PROGRAM S01_Loading
VAR
	//工站
	station					: REFERENCE TO FB_Station:=fbstation[1];
	//气缸
		fbVTCPressCyl_1	:REFERENCE TO FB_Cylinder:=fbCylinder[1];	//	链板线-下压气缸1
		fbVTCPressCyl_2	:REFERENCE TO FB_Cylinder:=fbCylinder[2];	//	链板线-下压气缸2
		fbVTCPressCyl_3	:REFERENCE TO FB_Cylinder:=fbCylinder[3];	//	链板线-下压气缸3
		fbVTCPressCyl_4	:REFERENCE TO FB_Cylinder:=fbCylinder[4];	//	链板线-下压气缸4
		fbVTCCyl_1	:REFERENCE TO FB_Cylinder:=fbCylinder[5];	//	移栽机构-Z轴气缸1
		fbVTCCyl_2	:REFERENCE TO FB_Cylinder:=fbCylinder[6];	//	移栽机构-Z轴气缸2
//链板线
		fbFlowLine:FB_FlowLine;	
		
	//伺服
		fbXAxisMove	 :REFERENCE TO FB_Axis:=fbAxis[1];	//	移栽上料X轴伺服
		fbYAxisMove	 :REFERENCE TO FB_Axis:=fbAxis[2];	//	移栽上料Y轴伺服
	//电动夹爪
		fbClamp_1:	 REFERENCE TO FB_ERG_20_Modbus:=fbERG_20_Modbus[1];
		fbClamp_2:	 REFERENCE TO FB_ERG_20_Modbus:=fbERG_20_Modbus[2];
	//相机
		 Camera   : 	 REFERENCE TO FB_Camera:=fbCamera[1]; 
	//延时
	arTonDelay :ARRAY[1..20] OF TON;
	//返回值
	UdiReturnValue :ARRAY[1..20] OF UDINT;
	//本地过程数据
	arProcessDataStation : ARRAY [1..2] OF DUT_MainlineFixture;
	//过程标志位
	xFlowLineReady:BOOL;//连班线准备流程完成信号
	xTakeBoxPremit:BOOL;//允许链板线执行下一循环
	//过程记录
	tsModuleProcess:ARRAY[1..gc_ModuleProNo] OF DUT_Process;
	xClearModuleProcessDone:BOOL;
	bClearProcessStep	:BYTE;
	
	
	i: INT;
	xFlowLineStart: BOOL;//链板线启动信号
	bFlowLineStep: BYTE;
	xFlowLineReadyCmd: BOOL;//连班线准备指令
	arFlowLineReachedSensor: ARRAY[1..4] OF BOOL;//链板线到位传感器
	_FirstFlag: ARRAY[1..10] OF BOOL;
	MachineInitR_TRIG:R_TRIG;

	// 程序循环
	bCounter: BYTE;
	// 上料工位到位传感器
	xLoadingReachedSensor: ARRAY[1..2] of bool;
	// 报警标志位
	_AlarmDisable: BOOL;
	// X轴放料循环
	bXCounter: BYTE;
	//夹爪有产品信号
	arClampHavePart :ARRAY[1..2] OF BOOL;
	iClearProcessStep: INT;
	// //首次循环
	_FirstCycle: ARRAY[1..10] of bool;
	//下压气缸原点传感器
	arVTCPressCylHPSensor:ARRAY[1..4] OF BOOL;
	//Y轴去放料位还是放料补偿位
	ariPosNum:ARRAY[1..2] OF INT;
	//下压气缸动点传感器
	arVTCPressCylWPSensor:ARRAY[1..4] OF BOOL;
	test: ARRAY[1..4]OF BOOL;
END_VAR

A_Input();
Alarm();
Delay();
FlowAuto();
FlowInit();
FlowLine();
General();
ILC();
TipAuto();
TipManual();
Z_Output();

ACTION A_Input:
//气缸
fbVTCPressCyl_1.xWP_Sensor	:=
arVTCPressCylWPSensor[1]		:=	IxS01VTCPressCyl_1WP 	;
fbVTCPressCyl_1.xHP_Sensor	:=
arVTCPressCylHPSensor[1]		:=	IxS01VTCPressCyl_1HP	;
fbVTCPressCyl_2.xWP_Sensor	:=	
arVTCPressCylWPSensor[2]		:=	IxS01VTCPressCyl_2WP	;
fbVTCPressCyl_2.xHP_Sensor	:=
arVTCPressCylHPSensor[2]		:=	IxS01VTCPressCyl_2HP	;
fbVTCPressCyl_3.xWP_Sensor	:=	
arVTCPressCylWPSensor[3]		:=IxS01VTCPressCyl_3WP	;
fbVTCPressCyl_3.xHP_Sensor	:=
arVTCPressCylHPSensor[3]		:=	IxS01VTCPressCyl_3HP	;
fbVTCPressCyl_4.xWP_Sensor	:=	
arVTCPressCylWPSensor[4]		:=IxS01VTCPressCyl_4WP	;
fbVTCPressCyl_4.xHP_Sensor	:=
arVTCPressCylHPSensor[4]		:=IxS01VTCPressCyl_4HP	;
fbVTCCyl_1.xWP_Sensor	:=	IxS01VTCCyl_1WP	;
fbVTCCyl_1.xHP_Sensor	:=	IxS01VTCCyl_1HP	;
fbVTCCyl_2.xWP_Sensor	:=	IxS01VTCCyl_2WP	;
fbVTCCyl_2.xHP_Sensor	:=	IxS01VTCCyl_2HP	;

//链板线传感器
arFlowLineReachedSensor[1]:=IxS01PositionSensor2;
arFlowLineReachedSensor[2]:=IxS01PositionSensor1;
arFlowLineReachedSensor[3]:=IxS01PositionSensor4;
arFlowLineReachedSensor[4]:=IxS01PositionSensor3;
//上料工位传感器
xLoadingReachedSensor[1]:=IxS01Sensor2Reached;
xLoadingReachedSensor[2]:=IxS01Sensor1Reached;
END_ACTION

ACTION Alarm:
//
station.adwAlarm[1].00:=station.xInitTimeout;	  //S01 初始化超时
(*station.adwAlarm[1].01:= //S01链板线上料位置1相机检测到深孔板放反，请检查
station.adwAlarm[1].02:=//S01链板线上料位置2相机检测到深放反，请检查
station.adwAlarm[1].03:=//S01链板线上料位置3相机检测到深孔板放反，请检查
station.adwAlarm[1].04:=//S01链板线上料位置4相机检测到深孔板放反，请检查
*)
station.adwAlarm[1].05	:=	fbClamp_1.eErrorID>24	;//	S01电动夹爪1报错，请检查
station.adwAlarm[1].06	:=	fbClamp_2.eErrorID>24	;//	S01电动夹爪2报错，请检查
//station.adwAlarm[1].07	:=	fbVTCPressCyl_1.xHP_Off 	;//	S01链板线-下压气缸1原点未到位
//station.adwAlarm[1].08	:=	fbVTCPressCyl_1.xWP_Off 	;//	S01链板线-下压气缸1动点未到位
//station.adwAlarm[1].09	:=	fbVTCPressCyl_2.xHP_Off	;//	S01链板线-下压气缸2原点未到位
//station.adwAlarm[1].10	:=	fbVTCPressCyl_2.xWP_Off	;//	S01链板线-下压气缸2动点未到位
//station.adwAlarm[1].11	:=	fbVTCPressCyl_3.xHP_Off	;//	S01链板线-下压气缸3原点未到位
//station.adwAlarm[1].12	:=	fbVTCPressCyl_3.xWP_Off	;//	S01链板线-下压气缸3动点未到位
//station.adwAlarm[1].13	:=	fbVTCPressCyl_4.xHP_Off	;//	S01链板线-下压气缸4原点未到位
//station.adwAlarm[1].14	:=	fbVTCPressCyl_4.xWP_Off	;//	S01链板线-下压气缸4动点未到位
station.adwAlarm[1].15	:=	fbVTCCyl_1.xHP_Off 	;//	S01移栽机构-Z轴气缸1原点未到位
station.adwAlarm[1].16	:=	fbVTCCyl_1.xWP_Off	;//	S01移栽机构-Z轴气缸1动点未到位
station.adwAlarm[1].17	:=	fbVTCCyl_2.xHP_Off 	;//	S01移栽机构-Z轴气缸2原点未到位
station.adwAlarm[1].18	:=	fbVTCCyl_2.xWP_Off	;//	S01移栽机构-Z轴气缸2动点未到位
station.adwAlarm[1].19	:=	fbXAxisMove.xError	;//	S01移栽上料X轴伺服报错
station.adwAlarm[1].20	:=	fbXAxisMove.xNotPowerOn	;//	S01移栽上料X轴伺服未使能
station.adwAlarm[1].21	:=	fbXAxisMove.xMoveTimeout	;//	S01移栽上料X轴伺服移动超时
station.adwAlarm[1].22	:=	fbYAxisMove.xError	;//	S01移栽上料Y轴伺服报错
station.adwAlarm[1].23	:=	fbYAxisMove.xNotPowerOn	;//	S01移栽上料Y轴伺服未使能
station.adwAlarm[1].24	:=	fbYAxisMove.xMoveTimeout	;//	S01移栽上料Y轴伺服移动超时
//station.adwAlarm[1].25	:=	fbFlowLine.xQError	;			//	S01移栽上料链板线报错

(*station.adwAlarm[1].26:= //S01链板线上料位置1相机检测到深孔板放反，请检查
station.adwAlarm[1].27:=//S01链板线上料位置2相机检测到深放反，请检查
station.adwAlarm[1].28:=//S01链板线上料位置3相机检测到深孔板放反，请检查
station.adwAlarm[1].29:=//S01链板线上料位置4相机检测到深孔板放反，请检查
*)
END_ACTION

ACTION Delay:
arTonDelay[01](IN:= , PT:=T#0.1S , Q=> , ET=> );
(*arTonDelay[02](IN:=  , PT:=T#1S , Q=> , ET=> );*)//链板线程序使用
arTonDelay[03](IN:=   , PT:=T#1S , Q=> , ET=> );
arTonDelay[04](IN:= , PT:=T#0.1S , Q=> , ET=> );
arTonDelay[05](IN:= , PT:=T#0.1S , Q=> , ET=> );
arTonDelay[06](IN:= , PT:=T#0.1S , Q=> , ET=> );
arTonDelay[07](IN:= , PT:=T#0.1S , Q=> , ET=> );
arTonDelay[08](IN:= NOT fbXAxisMove.xbusy , PT:=T#0.1S , Q=> , ET=> );//TipAuto使用
arTonDelay[09](IN:= NOT fbYAxisMove.xbusy, PT:=T#0.1S , Q=> , ET=> );//TipAuto使用
END_ACTION

ACTION FlowAuto:

//-----------------------------------------初始化是否完成判断----------------------------------------------
IF NOT station.xInitDone THEN
 	station.iStepAuto:=0;
 	station.xDone:=FALSE;
ELSIF station.xRunning  THEN
//-----------------------------------------动作步骤--------------------------------------------------------
CASE station.iStepAuto OF	  
	0: //----Home Step，等待启动----
		IF station.xDisabled 
			AND station.xCanRun 
			AND NOT fbMachine[1].xStopped 
			AND NOT station.xSingleRunning 
		THEN
			station.xDone:=TRUE;
		END_IF
		IF  station.xSingleRunning 
			OR station.xCanRun 
			//AND NOT station.xDone 
			AND NOT station.xDisabled 
			AND NOT fbMachine[1].xStopped
		THEN
			station.xCycleEnable:=TRUE;
			//station.xDone:= FALSE;  
			station.iStepAuto:= 10;
		END_IF
	10://复位
			Camera.xlInit:=TRUE;
			FOR  i:=1 TO  4 BY  1 DO
		 		sCamera_To_Plc.iS01Result[i]:=0;
			END_FOR
			MEMSET(ADR(arProcessDataStation[1]),0,SIZEOF(arProcessDataStation[1]));
			MEMSET(ADR(arProcessDataStation[2]),0,SIZEOF(arProcessDataStation[2]));
		
				 FOR i:=1 TO gc_ModuleProNo BY 1 DO
						 MEMSET(ADR(tsModuleProcess[i]),0,SIZEOF(tsModuleProcess[i]));
				 END_FOR
			station.iStepAuto:= 20;
  	20://此处开始处理上料流程
		station.iStepAuto:= 40;
//	30://Restore_after_Estop_Process1-拍照流程
//			IF  axBypassSignal[1] OR fbMachine[1].xTryRun THEN
//					station.iStepAuto :=110 ;
//			ELSIF tsModuleProcess[1].xProcessNotStarted AND NOT  tsModuleProcess[1].xProcessStarted THEN
//					station.iStepAuto :=40 ; (*process not started*)
//			ELSIF  tsModuleProcess[1].xProcessStarted AND NOT  tsModuleProcess[1].xProcessCompleted THEN
//				 station.iStepAuto :=40 ;(*process started*)
//			ELSIF  tsModuleProcess[1].xProcessCompleted AND NOT tsModuleProcess[1].xQDataCompleted  THEN
//					station.iStepAuto := 100 ;(*process completed*)
//			ELSIF tsModuleProcess[1].xQDataCompleted THEN
//					station.iStepAuto :=110 ;(*Qdata completed *)
//			ELSE    
//					station.iStepAuto :=40; 
//			END_IF
	40://启动链板线
		tsModuleProcess[1].xProcessNotStarted:=TRUE;
		fbFlowLine.xIRunningPremit:=TRUE;
			station.iStepAuto:=45;	
	45://链板线已启动
		IF   fbFlowLine.xQBusy THEN
		 		fbFlowLine.xIRunningPremit:=FALSE;
				station.iStepAuto:=50;	
		END_IF
	50://等待链板线执行结束
		IF 		NOT fbFlowLine.xQBusy THEN
		 		station.iStepAuto:=60;	
		END_IF
	60://Y轴去拍照位置
		fbYAxisMove.xMoveAuto[2]:=TRUE;
		IF  fbYAxisMove.xMoveInPos[2] THEN
		  	 station.iStepAuto:=70;	
		END_IF
	70://相机触发
		tsModuleProcess[1].xProcessStarted:=TRUE;
			Camera.xlTrigger:=TRUE;
			IF    Camera.xQBusy THEN
				Camera.xlTrigger:=FALSE;
				station.iStepAuto:=80;	
			END_IF
	80://等待相机完成
		IF  NOT Camera.xQBusy THEN
			station.iStepAuto:=100;		
		END_IF
		tsModuleProcess[1].xProcessCompleted:=TRUE;
	100://查看相机结果，判断是否料反
		(*位置1*)		
		_AlarmDisable:=FALSE;
		FOR  i:=1 TO 4 BY 1 DO
			IF 	sCamera_TO_Plc.iS01Result[i] >=3 THEN
					station.iStepAuto:=101;
					EXIT;
			ELSIF	i =4 THEN
					station.iStepAuto:=110;
			END_IF
		END_FOR
	101://报警,人工处理后重新拍照
		IF  NOT  _AlarmDisable THEN
					IF   sCamera_TO_Plc.iS01Result[1] =3 (*料反*) THEN
						station.adwAlarm[1].01:=TRUE ;//S01链板线上料位置1相机检测到深孔板放反，请检查
					ELSIF  sCamera_TO_Plc.iS01Result[1] =4 (*无料*) THEN
					 	station.adwAlarm[1].26:=TRUE ;//S01链板线上料位置1相机未检测到深孔板，请检查
					END_IF
					IF   sCamera_TO_Plc.iS01Result[2] =3 (*料反*) THEN
						station.adwAlarm[1].02:=TRUE ;//S01链板线上料位置2相机检测到深孔板放反，请检查
					ELSIF  sCamera_TO_Plc.iS01Result[2] =4 (*无料*) THEN
					 	station.adwAlarm[1].27:=TRUE ;//S01链板线上料位置2相机未检到板，请检查
					END_IF	
					IF   sCamera_TO_Plc.iS01Result[3] =3 (*料反*) THEN
 						station.adwAlarm[1].03:= TRUE;//S01链板线上料位置3相机检测到深孔板放反，请检查
					ELSIF  sCamera_TO_Plc.iS01Result[3] =4 (*无料*) THEN
					 	station.adwAlarm[1].28:=TRUE ;//S01链板线上料位置3相机未检到板，请检查
					END_IF
					IF    sCamera_TO_Plc.iS01Result[4] =3 (*料反*) THEN
 						station.adwAlarm[1].04:= TRUE;//S01链板线上料位置4相机检测到深孔板放反，请检查
					ELSIF  sCamera_TO_Plc.iS01Result[4] =4 (*无料*) THEN
					 	station.adwAlarm[1].29:=TRUE ;//S01链板线上料位置4相机未检到板，请检查
					END_IF
					_AlarmDisable:=TRUE;
		END_IF
			station.iStepAuto:=60;
	110://数据传送完成
			tsModuleProcess[1].xQDataCompleted:=TRUE;
			station.iStepAuto:=150;

///预留复检步骤120-150
	150://开始循环。循环次数=2
		IF NOT  fbMachine[1].xTryRun THEN
				IF  arFlowLineReachedSensor[1] AND arFlowLineReachedSensor[3]   THEN
								bCounter:=1;
								station.iStepAuto :=170; 
				ELSIF arFlowLineReachedSensor[2] AND arFlowLineReachedSensor[4] THEN
								bCounter:=2;
								station.iStepAuto :=170; 
				ELSE
								station.iStepAuto :=999; 
				END_IF
				
		ELSE
				 IF   NOT _FirstFlag[2] THEN
						bCounter:=1;
						_FirstFlag[2]:=TRUE;
				END_IF
		 		station.iStepAuto :=170; 
		END_IF
//	160://Restore_after_Estop_Process2/3 取孔板流程1/2
//			IF  station.xSingleRunning OR fbMachine[1].xTryRun THEN
//					station.iStepAuto :=170; 
//			ELSIF tsModuleProcess[bCounter+1].xProcessNotStarted AND NOT  tsModuleProcess[bCounter+1].xProcessStarted THEN
//					station.iStepAuto :=190 ; (*process not started*)
//			ELSIF  tsModuleProcess[bCounter+1].xProcessStarted AND NOT  tsModuleProcess[bCounter+1].xProcessCompleted THEN
//				 station.iStepAuto :=185 ;(*process started*)
//			ELSIF  tsModuleProcess[bCounter+1].xProcessCompleted AND NOT tsModuleProcess[bCounter+1].xQDataCompleted  THEN
//					station.iStepAuto := 230 ;(*process completed*)
//			ELSE
//					station.iStepAuto :=170; 
//			END_IF
	170://
			tsModuleProcess[bCounter+1].xProcessNotStarted :=TRUE;
			 station.iStepAuto:=190;
//		(***异常处理开始*)
//	185://电动夹爪打开
//			fbClamp_1.aReleaseControl[1]:=TRUE;
//			fbClamp_2.aReleaseControl[1]:=TRUE;
//			IF fbClamp_1.xDone  AND fbClamp_2.xDone   THEN
//					fbClamp_1.xExecute :=FALSE ;
//					fbClamp_2.xExecute:=FALSE;
//					 station.iStepAuto:=166;
//			END_IF	
//	186://Z轴上升
//			fbVTCCyl_1.xAuto:=FALSE;
//			fbVTCCyl_2.xAuto:=FALSE;
//		IF  fbVTCCyl_1.xHP_Delay AND 
//			fbVTCCyl_2.xHP_Delay THEN
//			 station.iStepAuto:=190;		
//		END_IF
//	(***异常处理结束*)			  
	190://XY轴去夹取位置1/2
			fbXAxisMove.xMoveAuto[bCounter +1]:=TRUE;
			fbYAxisMove.xMoveAuto[3]:=TRUE;
			fbClamp_1.aRotateReleaseControl[1]:=TRUE ;
			fbClamp_2.aRotateReleaseControl[1]:=TRUE ;		
			IF fbXAxisMove.xMoveInPos[bCounter+1] AND 
			   fbYAxisMove.xMoveInPos[3] AND 
				 fbClamp_1.xDone AND  
			  fbClamp_2.xDone THEN
					fbClamp_1.xExecute :=FALSE ;
				 fbClamp_2.xExecute :=FALSE ;
				 station.iStepAuto:=200;	
			END_IF
			
	200://Z轴气缸下降
		fbVTCCyl_1.xAuto:=TRUE;
		fbVTCCyl_2.xAuto:=TRUE;
		IF  fbVTCCyl_1.xWP_Delay AND 
			fbVTCCyl_2.xWP_Delay THEN
			 station.iStepAuto:=210;		
		END_IF
	210://电动夹爪夹取
				tsModuleProcess[bCounter+1].xProcessStarted :=TRUE;
		IF  fbmachine[1].xTryRun THEN 
				station.iStepAuto:=220;	
		ELSE
			fbClamp_1.aClampControl[1]:=TRUE;
			fbClamp_2.aClampControl[1]:=TRUE;
			IF (fbClamp_1.xDone OR (fbClamp_1.xGripClampEmpty  AND fbMachine[1].xTryRun)) AND
			 (fbClamp_2.xDone OR (fbClamp_2.xGripClampEmpty  AND fbMachine[1].xTryRun ))   THEN
					fbClamp_1.xExecute :=FALSE ;
					fbClamp_2.xExecute:=FALSE;
					 station.iStepAuto:=220;	
			END_IF
		END_IF	 
	220://Z轴上升
			arClampHavePart[1]:=TRUE;//夹爪1有产品标志位
			arClampHavePart[2]:=TRUE;//夹爪2有产品标志位
			tsModuleProcess[bCounter+1].xProcessCompleted :=TRUE;
				fbVTCCyl_1.xAuto:=FALSE;
				fbVTCCyl_2.xAuto:=FALSE;
			IF  fbVTCCyl_1.xHP_Delay AND 
				fbVTCCyl_2.xHP_Delay THEN
				 station.iStepAuto:=225;		
			END_IF
	225://判断流程
			IF bCounter =2 THEN
					xTakeBoxPremit:=TRUE;//允许链板线执行动作
			END_IF
			station.iStepAuto:=240;	
//	230://Restore_after_Estop_Process4 /Process5翻转孔板流程1/2
//			IF  station.xSingleRunning OR fbMachine[1].xTryRun THEN
//					station.iStepAuto :=240; 
//			ELSIF tsModuleProcess[bCounter+3].xProcessNotStarted AND NOT  tsModuleProcess[bCounter+3].xProcessStarted THEN
//					station.iStepAuto :=240 ; (*process not started*)
//			ELSIF  tsModuleProcess[bCounter+3].xProcessStarted AND NOT  tsModuleProcess[bCounter+3].xProcessCompleted THEN
//				 station.iStepAuto :=240;(*process started*)
//			ELSIF  tsModuleProcess[bCounter+3].xProcessCompleted AND NOT tsModuleProcess[bCounter+3].xQDataCompleted  THEN
//					station.iStepAuto :=280 ;(*process completed*)
//			ELSE
//					station.iStepAuto :=240; 
//			END_IF
	
	240://判断是否需要翻转
			IF  NOT  fbmachine[1].xTryRun THEN
			 		IF   bCounter =1 THEN
					 			IF 	sCamera_To_Plc.iS01Result[2] =2(*角度反*) OR sCamera_To_Plc.iS01Result[4] =2(*角度反*) THEN 
													 station.iStepAuto:=250;
								ELSE
								 							ariPosNum[1]:=4	;	
															ariPosNum[2]:=4	;	
														 station.iStepAuto:=280;			
								END_IF
								
					ELSIF  bCounter =2 THEN
					 			IF 	sCamera_To_Plc.iS01Result[1] =2(*角度反*) OR sCamera_To_Plc.iS01Result[3] =2(*角度反*) THEN 
													 station.iStepAuto:=250;
								ELSE
								 							ariPosNum[1]:=4	;	
															ariPosNum[2]:=4	;	
														 station.iStepAuto:=280;			
								END_IF
	
					END_IF
			ELSE
			 							station.iStepAuto:=280;			
			END_IF
	250://去翻转位
						tsModuleProcess[bCounter+3].xProcessNotStarted :=TRUE;
			 		 fbXAxisMove.xMoveAuto[6]:=TRUE;
					IF fbXAxisMove.xMoveInPos[6] THEN
						 station.iStepAuto:=260;	
					END_IF 	
  260://空跑
					tsModuleProcess[bCounter+3].xProcessStarted :=TRUE;
					station.iStepAuto:=265;	
	//261://判断夹爪是否需要调整
	//		IF  NOT xRotateCompletedClamp[1] AND NOT xRotateCompletedClamp[2] THEN
	//			station.iStepAuto:=265;
	//		ELSIF xRotateCompletedClamp[1] AND NOT xRotateCompletedClamp[2] THEN
	//			station.iStepAuto:=270;
	//		ELSIF  xRotateCompletedClamp[1] AND  xRotateCompletedClamp[2] THEN
	//			station.iStepAuto:=280;	
	//		END_IF
	265://夹爪1开始校正
				IF  (sCamera_To_Plc.iS01Result[1] =2(*角度反*) AND bCounter =2 ) OR
						(sCamera_To_Plc.iS01Result[2] =2(*角度反*) AND bCounter =1 ) THEN	
							fbClamp_1.aRotateClampControl[1]:=TRUE ;
							 IF (fbClamp_1.xDone OR (fbClamp_1.xClosecoverFailure AND fbmachine[1].xTryRun)) THEN						
									fbClamp_1.xExecute :=FALSE ;
									station.iStepAuto:= 270;
							END_IF
						ariPosNum[1]:=6	;	
				ELSE
				 		ariPosNum[1]:=4	;	
				 		station.iStepAuto:= 270;
				END_IF
	270://夹爪2开始校正			
				IF  (sCamera_To_Plc.iS01Result[3] =2(*角度反*) AND bCounter =2 ) OR
						(sCamera_To_Plc.iS01Result[4] =2(*角度反*) AND bCounter =1 ) THEN
						fbClamp_2.aRotateClampControl[1]:=TRUE ;
						 IF (fbClamp_2.xDone OR (fbClamp_2.xClosecoverFailure AND fbmachine[1].xTryRun)) THEN			
									fbClamp_2.xExecute :=FALSE ;
									station.iStepAuto:= 280;
							END_IF		
								ariPosNum[2]:=6	;	
				ELSE	
				 				ariPosNum[2]:=4	;	
				 				station.iStepAuto:= 280;
				END_IF	
	280://夹爪矫正完成
			tsModuleProcess[bCounter+3].xProcessCompleted:=TRUE;
			station.iStepAuto:=285;
	285://检查是否允许放料
			IF  NOT  xLoadingReachedSensor[1]  AND
				NOT  xLoadingReachedSensor[2]  AND 
			(( NOT station.xDone 			   AND
			 (NOT _FirstCycle[4] OR  S08_Mainline.station.xDone)) OR station.xSingleRunning) THEN
				 station.iStepAuto:=290;
				 _FirstCycle[4]:=TRUE;
		 END_IF
			
	290://X轴放料开始循环计数  =2
			IF ( bXCounter >2) OR NOT _FirstCycle[2] THEN
		 		bXCounter:=1;
				_FirstCycle[2]:=TRUE;
			END_IF
			station.iStepAuto :=300;
	295://Restore_after_Estop_Process6/7 孔板放料流程1/2
//			IF  station.xSingleRunning OR fbMachine[1].xTryRun THEN
//					station.iStepAuto :=300; 
//			ELSIF tsModuleProcess[bXCounter+5].xProcessNotStarted AND NOT  tsModuleProcess[bXCounter+5].xProcessStarted THEN
//					station.iStepAuto :=300 ; (*process not started*)
//			ELSIF  tsModuleProcess[bXCounter+5].xProcessStarted AND NOT  tsModuleProcess[bXCounter+5].xProcessCompleted THEN
//				 station.iStepAuto :=300;(*process started*)
//			ELSIF  tsModuleProcess[bXCounter+5].xProcessCompleted AND NOT tsModuleProcess[bXCounter+5].xQDataCompleted  THEN
//					station.iStepAuto :=330;(*process completed*)
//			ELSE
//					station.iStepAuto :=300; 
//			END_IF	
			station.iStepAuto :=300; 
	300://X轴去放料位置	
			tsModuleProcess[bXCounter+5].xProcessNotStarted:=TRUE;
			IF   bXCounter=1 THEN
						fbXAxisMove.xMoveAuto[4]:=TRUE;
						fbYAxisMove.xMoveAuto[ariPosNum[2]]:=TRUE;
								IF fbXAxisMove.xMoveInPos[4] AND 
									 fbYAxisMove.xMoveInPos[ariPosNum[2]] THEN
											 station.iStepAuto:=310;	
								END_IF				
			ELSIF	 bXCounter=2 THEN
			 			 fbXAxisMove.xMoveAuto[5]:=TRUE;
						 fbYAxisMove.xMoveAuto[ariPosNum[1]]:=TRUE;
								IF fbXAxisMove.xMoveInPos[5] AND 
									 fbYAxisMove.xMoveInPos[ariPosNum[1]] THEN
											 station.iStepAuto:=310;
								END_IF				
			END_IF
	310://Z轴下降
				IF   bXCounter=1 THEN
						fbVTCCyl_2.xAuto:=TRUE;
						IF fbVTCCyl_2.xWP_Delay THEN
							 station.iStepAuto:=320;	
						END_IF
				ELSIF	 bXCounter=2 THEN
								fbVTCCyl_1.xAuto:=TRUE;
						IF fbVTCCyl_1.xWP_Delay THEN
							 station.iStepAuto:=320;	
						END_IF					
			END_IF
	320://电动夹爪松开
			tsModuleProcess[bXCounter+5].xProcessStarted:=TRUE;
		//	IF  NOT  fbMachine[1].xTryRun THEN
				IF   bXCounter=1 THEN
								fbClamp_2.aReleaseControl[1]:=TRUE;
							IF fbClamp_2.xDone THEN
								fbClamp_2.xExecute:=FALSE;
								 station.iStepAuto:=330;	
							END_IF				
				ELSIF	 bXCounter=2 THEN
							fbClamp_1.aReleaseControl[1]:=TRUE;
							IF fbClamp_1.xDone THEN
								fbClamp_1.xExecute:=FALSE;
								 station.iStepAuto:=330;	
							END_IF			
				END_IF		
		//	ELSE
		//	  	station.iStepAuto:=330;	
		//	 END_IF
	330://传感器检测
				tsModuleProcess[bXCounter+5].xProcessCompleted:=TRUE;
				arClampHavePart[bXCounter]:=FALSE;//夹爪1/2有产品标志位
				IF   xLoadingReachedSensor[bXCounter] OR fbMachine[1].xTryRun THEN
					station.iStepAuto:=340;	
				END_IF
	340://Z轴上升		
				IF   bXCounter=1 THEN
							fbVTCCyl_2.xAuto:=FALSE;
						IF fbVTCCyl_2.xHP_Delay THEN
							 station.iStepAuto:=350;	
						END_IF	
				ELSIF	 bXCounter=2 THEN
							fbVTCCyl_1.xAuto:=FALSE;
						IF fbVTCCyl_1.xHP_Delay THEN
							 station.iStepAuto:=350;	
						END_IF				
				END_IF
	350://Restore_after_Estop_Process8 数据传输流程
			 IF  station.xSingleRunning THEN//OR fbMachine[1].xTryRun THEN
					 station.iStepAuto :=400; 
			ELSIF tsModuleProcess[8].xProcessNotStarted AND NOT  tsModuleProcess[8].xProcessStarted THEN
					 station.iStepAuto :=360; (*process not started*)
			 ELSIF  tsModuleProcess[8].xProcessStarted AND NOT  tsModuleProcess[8].xProcessCompleted THEN
					station.iStepAuto :=370;(*process started*)
			 ELSIF  tsModuleProcess[8].xProcessCompleted AND NOT tsModuleProcess[8].xQDataCompleted  THEN
					 station.iStepAuto :=400 ;(*process completed*)
			 ELSE
					 station.iStepAuto :=360; 
			 END_IF		
		 
	360://任务成功
		 tsModuleProcess[8].xProcessNotStarted:=TRUE;
		 tsModuleProcess[8].xProcessStarted:=TRUE;
		 
		 arProcessDataStation[1].xMaterialOnOff:=TRUE;
		 arProcessDataStation[2].xMaterialOnOff:=TRUE;
		 
		 arProcessDataStation[1].stProduct.xLoading_OK:=TRUE;
		 arProcessDataStation[2].stProduct.xLoading_OK:=TRUE;
		 station.iStepAuto:= 370;
	370://数据unload
			 MEMCPY(ADR(arMainlineFixtureData[arCurFixtureNumStation[1]]),ADR(arProcessDataStation[1]),SIZEOF(arProcessDataStation[1]));
			 MEMCPY(ADR(arMainlineFixtureData[arCurFixtureNumStation[2]]),ADR(arProcessDataStation[2]),SIZEOF(arProcessDataStation[2]));
			 station.iStepAuto:= 380;
	380://本地数据清除
			 	FOR i:=1 TO gc_ModuleProNo BY 1 DO
				 MEMSET(ADR(tsModuleProcess[i]),0,SIZEOF(tsModuleProcess[i]));
			 END_FOR
			 tsModuleProcess[8].xProcessCompleted:=TRUE;
			 station.iStepAuto:= 400;		
			 
			
	400://放料完成
			IF bXCounter =2 THEN
				station.xDone:=TRUE;
			END_IF
			station.iStepAuto:=420;
	//410://夹爪旋转回原位置
	//		IF NOT  fbMachine[1].xTryRun THEN
	//				IF   bXCounter=1 THEN
	//								 fbClamp_2.aRotateReleaseControl[1]:=TRUE ;
	//							IF fbClamp_2.xDone THEN
	//								 fbClamp_2.xExecute :=FALSE ;
	//								 station.iStepAuto:=420;	
	//							END_IF	
	//					ELSIF	 bXCounter=2 THEN
	//								fbClamp_1.aRotateReleaseControl[1]:=TRUE ;		
	//							IF fbClamp_1.xDone THEN
	//								 fbClamp_1.xExecute :=FALSE ;
	//								 station.iStepAuto:=420;	
	//							END_IF				
	//				END_IF
	//	ELSE	
	//	 			 station.iStepAuto:=420;	
	//	END_IF
	420://X轴循环+1
			bXCounter :=bXCounter +1;
			station.iStepAuto:=430;	

	430:  
		IF   bXCounter<=2 THEN
				station.iStepAuto:=295;	
		ELSE
				station.iStepAuto:=440;	
		END_IF

	440://循环-1
	IF  fbMachine[1].xTryRun THEN
			bCounter :=bCounter +1;
			station.iStepAuto:=450;
	ELSE
	 		station.iStepAuto:=150;
	END_IF
		
	450://空运行使用
		IF 	 bCounter <=2 THEN
			 station.iStepAuto:=160;	
		ELSE
		 	  station.iStepAuto:=999;
		END_IF
	999://----Single Run Finish----
		station.iStepAuto :=0;
		station.xSingleRunFlag:=FALSE;
		station.xCycleEnable:=FALSE;	
	//	station.xDone:=TRUE;

	ELSE
		;	
END_CASE

END_IF
END_ACTION

ACTION FlowInit:
IF NOT station.xIniting THEN
  station.iStepInit:=0;    

ELSE
//--------------------------------------------初始化步序----------------------------------
CASE station.iStepInit OF	
 0://  
  	IF station.xIniting THEN	
  	  station.iStepInit:=10;	
  	END_IF	
10://复位数据
		FOR i:=1 TO gc_ModuleProNo BY 1 DO
				MEMSET(ADR(tsModuleProcess[i]),0,SIZEOF(tsModuleProcess[i]));
		END_FOR
		FOR  i:=1 TO  4 BY  1 DO
		 		sCamera_To_Plc.iS01Result[i]:=0;
		END_FOR
		fbClamp_1.xInitControl:=FALSE;
		fbClamp_1.xInitControl:=FALSE ;
		fbClamp_1.xExecute :=FALSE;
		fbClamp_2.xExecute:=FALSE;
		IF NOT fbMachine[1].xTryRun THEN
				Camera.xlInit:=TRUE;
		END_IF
    station.iStepInit := 20;
20://Z轴上升
	 fbVTCCyl_1.xinit := TRUE; 
	 fbVTCCyl_2.xInit:=TRUE;
	IF fbVTCCyl_1.xHP_Delay AND fbVTCCyl_2.xHP_Delay  THEN
    		station.iStepInit:=40;	
	END_IF		
40: //伺服上电
  	 fbXAxisMove.xPowerInit := TRUE ;
	 fbYAxisMove.xPowerInit := TRUE ;
	IF fbXAxisMove.xPowerOn AND   fbYAxisMove.xPowerOn THEN 
    	station.iStepInit:=50;	
	END_IF
50://伺服去待机位置
		fbXAxisMove.xMoveAuto[1]:=TRUE;
		fbYAxisMove.xMoveAuto[1]:=TRUE;
		IF fbXAxisMove.xMoveInPos[1] AND fbYAxisMove.xMoveInPos[1]  THEN
			station.iStepInit:=60;	
		END_IF
60://电动夹爪初始化
	//	IF    NOT    arClampHavePart[1]  THEN
				fbClamp_1.xInitControl:=TRUE ;
	//	END_IF
	//	IF    NOT    arClampHavePart[2]  THEN
				 fbClamp_2.xInitControl:=TRUE ;
	//	END_IF
		 IF  (fbClamp_1.xDone (*OR  arClampHavePart[1]*) )   AND 
			 (fbClamp_2.xDone (*OR  arClampHavePart[2]*) ) THEN 
			fbClamp_1.xExecute :=FALSE;
			fbClamp_2.xExecute:=FALSE;
			station.iStepInit:=70;
		 END_IF				
70://电动夹爪去初始位置
				fbClamp_1.aReleaseControl[1]:=TRUE ;
				fbClamp_2.aReleaseControl[1]:=TRUE ;
		 IF  fbClamp_1.xDone AND fbClamp_2.xDone THEN 
			fbClamp_1.xExecute :=FALSE;
			fbClamp_2.xExecute:=FALSE;
			station.iStepInit:=80;
		 END_IF						
80://链板线初始化
		fbFlowLine.xIInit:=TRUE;
		station.iStepInit:=90;
90://等待完成
		IF  NOT fbFlowLine.xQBusy THEN
			 	station.iStepInit:=100;
		END_IF
100://
       station.iStepInit:=999;	

999://初始化完成	
	station.iStepInit:=0;
	station.xInitDone:=TRUE;  
END_CASE
END_IF
END_ACTION

ACTION FlowLine:
	
	fbFlowLine(
	arIReachedSensor:= arFlowLineReachedSensor,
	arIVTCCylHPSensor:=arVTCPressCylHPSensor , 
	arIVTCCylWPSensor:=arVTCPressCylWPSensor , 
	xIRunningPremit:= ,
	xIInit:= station.xIniting,
	xIEmptyDone:=  fbMachine[1].xEmptyDone, 
	xITryRun:= fbMachine[1].xTryRun, 
	xIMotorEstop:=  not  fbMachine[1].xEStop, 
	xIMotorStartButtonHmi:=arFlowLineControl[1] , 
	xIMotorStopButtonHmi:= arFlowLineControl[2], 
	xIManualMode:= fbMachine[1].xManualMode , 
	xIAutoMode:= fbMachine[1].xAutoMode, 
	arQVTCCylHPValve=> , 
	arQVTCCylWPValve=> , 
	xQMotorEstop=> QxFlowLineSpeedCtrl_1, 
	xQMotorStop=> QxFlowLineStop, 
	xQMotorStart=>QxFlowLineStart , 
	xQBusy=> , 
	xQError=> );
END_ACTION

ACTION General:
MachineInitR_TRIG(CLK:=fbMachine[1].xInitDone , Q=> );
IF  MachineInitR_TRIG.Q THEN
	_FirstCycle[4]:=FALSE;
END_IF
END_ACTION

ACTION ILC:

//---------------------------------------------------工站可执行-------------------------------------------------------
station.xCanRun := TRUE ;

//---------------------------------------------------气缸动作条件-------------------------------------------
fbVTCPressCyl_1.xOffILC	:=	TRUE	;
fbVTCPressCyl_1.xOnILC	:=	TRUE	;
fbVTCPressCyl_2.xOffILC	:=	TRUE	;
fbVTCPressCyl_2.xOnILC	:=	TRUE	;
fbVTCPressCyl_3.xOffILC	:=	TRUE	;
fbVTCPressCyl_3.xOnILC	:=	TRUE	;
fbVTCPressCyl_4.xOffILC	:=	TRUE	;
fbVTCPressCyl_4.xOnILC	:=	TRUE	;
fbVTCCyl_1.xOffILC	:=	TRUE	;
fbVTCCyl_1.xOnILC	:=	TRUE	;
fbVTCCyl_2.xOffILC	:=	TRUE	;
fbVTCCyl_2.xOnILC	:=	TRUE	;



//---------------------------------------------------伺服动作条件-------------------------------------------
fbXAxisMove.xRunILC 	:= 		
fbXAxisMove.xMoveILC[1]	:= 		
fbXAxisMove.xMoveILC[2] 	:= 		
fbXAxisMove.xMoveILC[3]	:= 		
fbXAxisMove.xMoveILC[4]	:= 		
fbXAxisMove.xMoveILC[5]	:= 
fbXAxisMove.xMoveILC[6]	:= 	fbVTCCyl_1.xHP_Sensor	AND 	fbVTCCyl_2.xHP_Sensor	;
fbYAxisMove.xRunILC 	:= 		
fbYAxisMove.xMoveILC[1]	:= 		
fbYAxisMove.xMoveILC[2]	:= 		
fbYAxisMove.xMoveILC[3]	:= 		
fbYAxisMove.xMoveILC[4]	:= 		
fbYAxisMove.xMoveILC[5]	:= 	fbVTCCyl_1.xHP_Sensor	AND 	fbVTCCyl_2.xHP_Sensor	;
///电动夹爪
fbERG_20_Modbus[1].xDeviceRunning:=
fbERG_20_Modbus[2].xDeviceRunning:=station.xSingleRunning OR station.xRunning OR station.xIniting;

Camera.xIDeviceRunning:=station.xSingleRunning;
END_ACTION

ACTION TipAuto:
//------------------------------------------------AutoTip Cylinder--------------------------------
//station.adwAutoTip[1].00	:=	fbVTCPressCyl_1.xAutoTip	;
//station.adwAutoTip[1].01	:=	fbVTCPressCyl_2.xAutoTip	;
//station.adwAutoTip[1].02	:=	fbVTCPressCyl_3.xAutoTip	;
//station.adwAutoTip[1].03	:=	fbVTCPressCyl_4.xAutoTip	;
station.adwAutoTip[1].04	:=	fbVTCCyl_1.xAutoTip	;
station.adwAutoTip[1].05	:=	fbVTCCyl_2.xAutoTip	;

//------------------------------------------------AutoTip Servo--------------------------------
//**************************************
FOR i:= 1 TO 5 BY 1 DO 
	IF fbXAxisMove.xMoveAuto[i] THEN
		fbXAxisMove.iPosNumber := i ;
	END_IF
	IF fbYAxisMove.xMoveAuto[i] THEN
		fbYAxisMove.iPosNumber := i ;
	END_IF
END_FOR
IF fbMachine[1].xAutoMode AND NOT fbMachine[1].xRunning  AND  arTonDelay[9].Q  THEN 
		IF fbXAxisMove.iPosNumber=1 AND NOT fbXAxisMove.xMoveInPos[1] THEN station.adwAutoTip[1].10:=TRUE; END_IF//轴伺服自动时位置不在位置1	
		IF fbXAxisMove.iPosNumber=2 AND NOT fbXAxisMove.xMoveInPos[2] THEN station.adwAutoTip[1].11:=TRUE; END_IF//轴伺服自动时位置不在位置2	
		IF fbXAxisMove.iPosNumber=3 AND NOT fbXAxisMove.xMoveInPos[3] THEN station.adwAutoTip[1].12:=TRUE; END_IF//轴伺服自动时位置不在位置3	
		IF fbXAxisMove.iPosNumber=4 AND NOT fbXAxisMove.xMoveInPos[4] THEN station.adwAutoTip[1].13:=TRUE; END_IF//轴伺服自动时位置不在位置4	
		IF fbXAxisMove.iPosNumber=5 AND NOT fbXAxisMove.xMoveInPos[5] THEN station.adwAutoTip[1].14:=TRUE; END_IF//轴伺服自动时位置不在位置5	
END_IF
IF fbMachine[1].xAutoMode AND NOT fbMachine[1].xRunning  AND  arTonDelay[10].Q  THEN 		
		
		IF fbYAxisMove.iPosNumber=1 AND NOT fbYAxisMove.xMoveInPos[1] THEN station.adwAutoTip[1].15:=TRUE; END_IF//轴伺服自动时位置不在位置1	
		IF fbYAxisMove.iPosNumber=2 AND NOT fbYAxisMove.xMoveInPos[2] THEN station.adwAutoTip[1].16:=TRUE; END_IF//轴伺服自动时位置不在位置2	
		IF fbYAxisMove.iPosNumber=3 AND NOT fbYAxisMove.xMoveInPos[3] THEN station.adwAutoTip[1].17:=TRUE; END_IF//轴伺服自动时位置不在位置3	
		IF fbYAxisMove.iPosNumber=4 AND NOT fbYAxisMove.xMoveInPos[4] THEN station.adwAutoTip[1].18:=TRUE; END_IF//轴伺服自动时位置不在位置4	
		IF fbYAxisMove.iPosNumber=5 AND NOT fbYAxisMove.xMoveInPos[5] THEN station.adwAutoTip[1].19:=TRUE; END_IF//轴伺服自动时位置不在位置5	
END_IF
END_ACTION

ACTION TipManual:
//--------------------------------------------ManualTip------------------------------------------------------

//-------------------------------------------气缸提示---------------------------------------------------------


//-------------------------------------------伺服提示--------------------------------------------------

/////////////////////////////////////////////////////////////////////////////////////////////////////////////////
END_ACTION

ACTION Z_Output:
(**************************气缸输出********************************)
QxS01VTCPressCyl_1WP	:=	(NOT  fbMachine[1].xAutoMode AND NOT station.xSingleRunning  AND    fbVTCPressCyl_1.xWP_Valve	) OR
												 ( (fbMachine[1].xAutoMode OR  station.xsingleRunning ) AND  	fbFlowLine.arQVTCCylWPValve[1]);
QxS01VTCPressCyl_1HP	:=	(NOT  fbMachine[1].xAutoMode AND NOT station.xSingleRunning  AND    fbVTCPressCyl_1.xHP_Valve	) OR
												 ( (fbMachine[1].xAutoMode OR  station.xsingleRunning ) AND  	fbFlowLine.arQVTCCylHPValve[1]);
QxS01VTCPressCyl_2WP	:=	(NOT  fbMachine[1].xAutoMode AND NOT station.xSingleRunning  AND    fbVTCPressCyl_2.xWP_Valve	) OR
												 ( (fbMachine[1].xAutoMode OR  station.xsingleRunning ) AND  	fbFlowLine.arQVTCCylWPValve[2]);
QxS01VTCPressCyl_2HP	:=	(NOT  fbMachine[1].xAutoMode AND NOT station.xSingleRunning  AND    fbVTCPressCyl_2.xHP_Valve	) OR
												 ( (fbMachine[1].xAutoMode OR  station.xsingleRunning ) AND  	fbFlowLine.arQVTCCylHPValve[2]);
QxS01VTCPressCyl_3WP	:=			(NOT  fbMachine[1].xAutoMode AND NOT station.xSingleRunning  AND    fbVTCPressCyl_3.xWP_Valve	) OR
												 ( (fbMachine[1].xAutoMode OR  station.xsingleRunning ) AND  	fbFlowLine.arQVTCCylWPValve[3]);
QxS01VTCPressCyl_3HP	:=	(NOT  fbMachine[1].xAutoMode AND NOT station.xSingleRunning  AND    fbVTCPressCyl_3.xHP_Valve	) OR
												 ( (fbMachine[1].xAutoMode OR  station.xsingleRunning ) AND  	fbFlowLine.arQVTCCylHPValve[3]);
QxS01VTCPressCyl_4WP	:=				(NOT  fbMachine[1].xAutoMode AND NOT station.xSingleRunning  AND    fbVTCPressCyl_4.xWP_Valve	) OR
												 ( (fbMachine[1].xAutoMode OR  station.xsingleRunning ) AND  	fbFlowLine.arQVTCCylWPValve[4]);
QxS01VTCPressCyl_4HP	:=		(NOT  fbMachine[1].xAutoMode AND NOT station.xSingleRunning  AND    fbVTCPressCyl_4.xHP_Valve	) OR
												 ( (fbMachine[1].xAutoMode OR  station.xsingleRunning ) AND  	fbFlowLine.arQVTCCylHPValve[4]);
QxS01VTCCyl_1WP	:=	fbVTCCyl_1.xWP_Valve	;
QxS01VTCCyl_1HP	:=	fbVTCCyl_1.xHP_Valve	;
QxS01VTCCyl_2WP	:=	fbVTCCyl_2.xWP_Valve	;
QxS01VTCCyl_2HP	:=	fbVTCCyl_2.xHP_Valve	;
END_ACTION

END_PROGRAM

(* stored: Version 1.1.0.1, ProductVersion 3.1.4024.9
   POU S01_Loading: Id {09eabbef-079c-4b02-9a4f-f15f03dbd456}, SpecialFunc None
   Action A_Input: Id {d02a1e8b-99f7-4a59-a9d7-b46699eb8bde}
   Action Alarm: Id {f91e2fff-b518-4309-9d5e-d947434883cd}
   Action Delay: Id {084f8558-cebd-455d-abdf-a99ad2ca1ee4}
   Action FlowAuto: Id {aff581fc-9b63-454d-b4be-e4b957bf91ee}
   Action FlowInit: Id {737815c3-3d44-47dd-9c07-561ee528fd92}
   Action FlowLine: Id {b28f4192-39f5-4366-9ebd-07d256861364}
   Action General: Id {853ea6bd-bb20-473d-996d-ff4ed10c4144}
   Action ILC: Id {0b3196e9-82f1-46a4-9b14-c04a89d888e7}
   Action TipAuto: Id {aecc5aff-b1ec-43bf-9301-a661c8b5dae6}
   Action TipManual: Id {561a1c1d-e3fd-42a1-bd5f-597305c6c45d}
   Action Z_Output: Id {f73574ac-bbd1-4517-bd7c-1b8c56ce8f05} *)
